{attribute 'Tc2GvlVarNames'}
VAR_GLOBAL
	arrLastAlarms: ARRAY [1..200] OF ST_AlarmStructure;
END_VAR

(* stored: Version 1.1.0.1, ProductVersion 3.1.4024.9
   GVL ArrLastAlarms: Id {2a3a34c6-215c-49d8-b2bd-e1ba95d6a24b} *)
